Staubli VAL3: page_Production.pjx

--- page_Production.pjx ---
Parameters version=s7.8.3 stackSize=5000 millimeterUnit=true
Program file=alreadyExist.pgx
Program file=buildList.pgx
Program file=cleanUserMenu.pgx
Program file=defineTraj.pgx
Program file=deleteItem.pgx
Program file=goTo.pgx
Program file=listAdd.pgx
Program file=loadPage.pgx
Program file=main.pgx
Program file=onEnterEvent.pgx
Program file=onExit.pgx
Program file=onF1Event.pgx
Program file=onF2Event.pgx
Program file=onF3Event.pgx
Program file=onF4Event.pgx
Program file=onF5Event.pgx
Program file=onF6Event.pgx
Program file=onF7Event.pgx
Program file=onF8Event.pgx
Program file=onLeftEvent.pgx
Program file=onRightEvent.pgx
Program file=onStart.pgx
Program file=refresh.pgx
Program file=refreshDynamic.pgx
Program file=refreshStatic.pgx
Program file=selectType.pgx
Program file=showStatus.pgx
Data file=page_Production.dtx
Library alias=data path=Disk://SaveData/SaveData.pjx
Library alias=pub path=Disk://public_temp/pub/pub.pjx
Library alias=use path=Disk://public_temp/userPage/userPage.pjx
Library alias=cycle path=Disk://cycle/cycle.pjx
Library alias=io path=Disk://io/io.pjx

--- page_Production.dtx ---
mdesc mNomSpeed
bool bTrigger
bool bShowStatus
bool bMoveRelease
bool bLarge
bool bButton[8]
  [4] = true
  [5] = true
  [6] = true
  [7] = true
num nClockStatus
num nIndex
num nKey = -1
num nIndexItem
num nOldIndex
public num nPage
num nRefresh = 2164.601
num nSelected
num nTime = 1
num nType
num nView
pointRx pPointTest[7]
string sEvent = "hello"
string sEventImport
string sImport
public string sItems
string sList = "hello"
string sMenu[8]
  [0] = "Simulation"
  [4] = "Type"
  [5] = "Duplicate"
  [6] = "Delete"
  [7] = "New"
string sMenu8[8]
string sMenuUser[8]
string sMessage
string sTrsfNum[8 6]
string sWorkingmode[8]

--- main.pgx ---
public program main()
  local bool l_bSave
  local bool l_bOverRide
  local bool l_bOk
  local bool l_bUnreached
  local string l_sMessage
begin
      // INIT
      call onStart()
        // LOOP UNTIL nKey=255
        nIndexItem=0
  do
    call refresh()
    nKey=getKey()
    call use:listevent(nKey,nIndex,sEvent)
    nView=use:nView
    switch nKey
      case 259
        // TAB
        bLarge=!bLarge
        //  call use:setView()
      break
      case 263
        // backSpace rename
        //call onBackEvent(l_bSave)
      break
      case 32
        // space to edit Action
        //call onSpaceEvent()
      break
      case 271
        call onF1Event()
      break
      case 272
        //
        call onF2Event()
      break
      case 273
        //
        call onF3Event()
      break
      case 274
        //
        call onF4Event()
      break
      case 275
        //
        call onF5Event()
      break
      //
      case 276
        call onF6Event()
      break
      case 277
        //
        call onF7Event()
      break
      case 278
        //
        call onF8Event()
      break
      case 270
        //
        call onEnterEvent()
      break
    endSwitch
    delay(0)
  until workingMode()!=4
      if workingMode()!=4 and workingMode()!=1
      call use:timerDialog("请切换至手动模式或者远程自动模式",0)
      wait(workingMode()==4 or workingMode()==1)
      delay(0)
     endIf
   use:bUseRefresh=true
      //  // exit
     call onExit(l_bSave)
end

--- buildList.pgx ---
program buildList()
  local num l_nSize
  local string l_sEvent
  local num i
  local bool l_bFound
  local num l_nCount
  local string l_sEmpty
  local num j
begin
    call use:stringCopy(l_sEmpty,sList)
  ////  call use:setSizeList(17,0,21,7)
  ////  call use:setSizeList(15,0,18,9)
  ////  建立对话款
  ////  call use:listcreate("")

  //  sWorkingmode[0]="[ ] 生产循环状态"
  //  sWorkingmode[1]="[ ] 循环暂停状态"
  //  sWorkingmode[2]="[ ] 机器人HOME点"
  //  sWorkingmode[3]="[ ] 机器人准备好"
  //  sWorkingmode[4]="[ ] 急停报警"
  //  sWorkingmode[5]="[ ] 防止碰撞功能开启"
  //  sWorkingmode[6]="[ ] 通讯正常"

  //  call use:listadd(sWorkingmode)
  //  call use:selectNewField(nSelected,nIndex,nView)
  //  call use:listupdate(0)
  // nIndex=data:nPage_Traj
  // call use:selectNewField(nSelected,nIndex,nView)
end

--- onEnterEvent.pgx ---
program onEnterEvent()
  local num i
  local num l_nIndex
  local string l_sItem[2]
  local num l_nResult
  local string l_sMessage
begin
  pub:libLoad("Disk://page/page_editTraj")
  call pub:main()
end

--- onF5Event.pgx ---
program onF5Event()
  local num i
  local num l_nValue
  local string l_sMessage
begin
//  // look if the bButton is enable
//  if bButton[4]
//    //
//    call selectType()
//    //
//    call buildList()
//    //
//    use:bUseRefresh=true
//  endIf
end

--- onF6Event.pgx ---
program onF6Event()
  local string l_sPaste
  local bool l_bUndo
  local num l_nResult
begin
//  // look if the bButton is enable
//  if bButton[5]
//    //
//    //  Duplicate
//    //
//    l_sPaste=sEvent
//    call alreadyExist(l_sPaste,l_bUndo)
//    if !l_bUndo
//      call trajType:duplicate(sEvent,l_sPaste,l_nResult)
//      if l_nResult==0
//        logMsg("[KERNEL] INTERFACE:Duplicate the trajectory: "+sEvent+" to: "+l_sPaste)
//        sEvent=l_sPaste
//        // update the memory stack
//        call buildList()
//      else
//        popUpMsg("error code duplicate: "+toString("",l_nResult))
//        logMsg("[KERNEL] INTERFACE:Duplicate the trajectory: "+sEvent+" to: "+l_sPaste+"errorCode"+toString("",l_nResult))
//      endIf
//    endIf
//  endIf
end

--- onF7Event.pgx ---
program onF7Event()
  local string l_sSwap
  local num l_nResult
  local string l_sMessage
  local string l_sMessage2
  local bool l_bYes
  local string l_sButton[2]
begin
//  // look if the bButton is enable
//  if bButton[6]
//    //
//    // delete a Trajectory
//    //
//    call deleteItem(l_bYes)
//    if l_bYes
//      call trajType:delete(sEvent,l_nResult)
//      if l_nResult==0
//        logMsg("[KERNEL] INTERFACE:Delete the trajectory: "+saveData:sTrajTypeUsing+" "+sEvent)
//        call buildList()
//      else
//        popUpMsg("error code: "+toString("",l_nResult))
//        logMsg("[KERNEL] INTERFACE:Delete the trajectory: "+saveData:sTrajTypeUsing+" "+sEvent+"error code: "+toString("",l_nResult))
//      endIf
//    endIf
//  endIf
end

--- onF8Event.pgx ---
program onF8Event()
  local string l_sNew
  local bool l_bUndo
  local num l_nResult
begin
//  // look if the bButton is enable
//  if bButton[7]
//    // new one
//    call alreadyExist(l_sNew,l_bUndo)
//    if !l_bUndo and l_sNew!=""
//      call trajType:new(l_sNew,l_nResult)
//      if l_nResult==0
//        logMsg("[KERNEL] INTERFACE:Create the new trajectory: "+saveData:sTrajTypeUsing+" "+l_sNew)
//        sEvent=l_sNew
//        call buildList()
//      else
//        popUpMsg("error code: "+toString("",l_nResult))
//        logMsg("[KERNEL] INTERFACE:Create the new trajectory: "+saveData:sTrajTypeUsing+" "+l_sNew+" error code "+toString("",l_nResult))
//      endIf
//    endIf
//  endIf
end

--- onRightEvent.pgx ---
program onRightEvent(bool& x_bSave)
  local num i
  local num l_nType
  local string l_sPath
  local string l_sEmpty
  local num l_nResult
  local string l_sMessage
begin
//  //
//  // right click
//  //
//  if x_bSave
//    x_bSave=false
//    l_sEmpty=""
//    l_nResult=0
//    call trajType:onSave(l_sEmpty)
//    // show the message
//    call language:message(l_sMessage,-4)
//    call use:timerDialog(l_sMessage,1)
//  endIf
//  // select the next one
//  do
//    nType=(nType+1)%(size(saveData:sTrajType))
//    saveData:sTrajTypeUsing=saveData:sTrajType[nType]
//    if saveData:sTrajType[nType]!=""
//      // find the good id
//      if saveData:sTrajType[nType]!=""
//        call saveData:getPathInstr(saveData:sTrajType[nType],l_sPath)
//      endIf
//    endIf
//  until saveData:sTrajType[nType]!=""
//  // load the type
//  if trajType:libPath()!=l_sPath and l_sPath!=""
//    i=trajType:libLoad(l_sPath)
//    delay(0)
//  endIf
//  if l_sPath==""
//    popUpMsg("error load traj type on ENTER "+saveData:sTrajTypeUsing+toString("",i))
//  endIf
//  // clean the user MENU
//  call cleanUserMenu()
//  // rebuild the list
//  call buildList()
end

--- onStart.pgx ---
program onStart()
  local num i
begin
  cls()
  userPage()
  call use:nullKey(nKey)
  call buildList()
    call refreshStatic()
 //   nRefresh=clock()
end

--- refresh.pgx ---
program refresh()
// // page refresh
begin
    if  (nKey>=270 and nKey<=278) or use:bUseRefresh==true
    call refreshStatic()
    call buildList()
    call refreshDynamic()
    if abs(clock()-nRefresh)>nTime
      call refreshDynamic()
    endIf
  endIf
end

--- refreshDynamic.pgx ---
program refreshDynamic()
  local string l_sMessage
  local string l_sItem
begin
//  // DO NOT CHANGE
  nRefresh=clock()
  use:bUseRefresh=false
  //  //
  if cycle:bCycle
    call use:type(18,1,"[X] 生产循环状态")
  else
    call use:type(18,1,"[ ] 生产循环状态")
  endIf

  if cycle:bPause
    call use:type(18,2,"[X] 生产循环暂停")
  else
    call use:type(18,2,"[ ] 生产循环暂停")
  endIf

  if cycle:bIsHome
    call use:type(18,3,"[X] 机器人Home电")
  else
    call use:type(18,3,"[ ] 机器人Home电")
  endIf

  if io:dOutIsReady==true
    call use:type(18,4,"[X] 机器人准备好")
  else
    call use:type(18,4,"[ ] 机器人准备好")
  endIf

  if cycle:bIsEstop
    call use:type(18,5,"[X] 急停报警")
  else
    call use:type(18,5,"[ ] 急停报警")
  endIf

  if io:dInCrashError==true
    call use:type(18,6,"[X] 防止碰撞开启信号")
  else
    call use:type(18,6,"[ ] 防止碰撞开启信号")
  endIf

  if cycle:bConnected_Plc
    call use:type(18,7,"[X] 通信正常")
  else
    call use:type(18,7,"[ ] 通信不正常")
  endIf
  call use:type(0,10,"现场运行程序项目-->"+io:sToShow+"                ")
end

--- refreshStatic.pgx ---
program refreshStatic()
  local string l_sMessage
  local num i
  local string l_sMenu
begin


   cls()
  //
  // set the view of the page..
  //
  // SET THE PAGE NUMBER
  use:nPage=0
  // USE <>PROFILE for <>PAGE

  // SET THE VIEW OF THE PAGE
  title("远程生产界面")
  //call language:page(l_sMenu,use:nPage)
//    l_sMenu="权限,,,,,吸片,放片,保存"
  // define the menu
  call use:stringToArray(l_sMenu,sMenu)
  // set the menu
  call use:setMenu(sMenu,false,1)
  call use:getMenu(sMenu,bButton)
  //
  // CREATE THE LIST
  //
  // define your list size for default
  call use:setSizeList(17,0,21,7)
 // call use:setSizeList(0,0,38,10)
  call use:setView(bLarge)
  //
  call use:listcreate("")
  //
  call use:listadd(sList)
  //
  // refresh the cursor
  use:nView=nView
  // refresh the list
  call use:listupdate(nIndex-nView)
end

--- selectType.pgx ---
program selectType()
  local string l_sMessage
  local num l_nIndex
  local string l_sEvent
  local num l_nKey
  local num i
  local string l_sPath
begin
//  // clean the line
//  call use:clear(0,13)
//  call language:message(l_sMessage,191)
//  call use:typeCenter(13,l_sMessage,40,true)
//  call use:setSizeList(15,2,10,6)
//  // TODO message
//  call use:listcreate("")
//  call use:listadd(saveData:sTrajType)
//  call use:selectNewField(nType,0,0)
//  // select the Item
//  do
//    l_nKey=get()
//    call use:listevent(l_nKey,l_nIndex,l_sEvent)
//  until l_nKey==270 or l_nKey==255
//  // choose the type
//  if l_nKey==270 and saveData:sTrajTypeUsing!=l_sEvent
//    saveData:sTrajTypeUsing=l_sEvent
//    // get the path
//    call saveData:getPathInstr(l_sEvent,l_sPath)
//    // load it
//    if trajType:libPath()!=l_sPath and l_sPath!=""
//      i=trajType:libLoad(l_sPath)
//      delay(0)
//    endIf
//    if l_sPath==""
//      popUpMsg("error load traj type on ENTER "+saveData:sTrajTypeUsing+toString("",i))
//    endIf
//  endIf
//  // clean the user MENU
//  call cleanUserMenu()
end
